TYPE "Positioning_MOL_Machine_Config"
VERSION : 0.1
// Block: Positioning_MOL_Machine_Config
   STRUCT
      DelayMissingCondition : Time;
      CyclicOBTime_ms : LReal;
      Ax : OOAx_Config;
      Ax_UM2 : udt_LinTranformation;
   END_STRUCT;

END_TYPE
